FUNCTION_BLOCK RunningToSuspendedUnifiedProgramTransition EXTENDS RunningToSuspendedProgramTransition
VAR_STAT
	//! <summary>Class name shared by all instances of this function block.</summary>
	{attribute 'OPC.UA.DA' := '0'}
	_ClassName : STRING := __POUNAME();
END_VAR

{attribute 'monitoring' := 'call'}
PROPERTY ClassName : REFERENCE TO STRING
GET
ClassName REF= _ClassName;
END_GET
END_PROPERTY

END_FUNCTION_BLOCK

(* stored: Version 1.1.0.1
   POU RunningToSuspendedUnifiedProgramTransition: Id {f0324d7c-cb47-4317-98ee-0ee523c67d2b}, SpecialFunc None
   Property ClassName: Id {e36aa9d5-f124-407e-bc42-b4e375b0f3e0}
   Get Get: Id {e15dc325-9d2e-424c-9cea-0526998166e7} *)
